{attribute 'linkalways'} 
{attribute 'no_explicit_call' := 'This FB is a CLASS and must be accessed using methods or properties'}
{attribute 'enable_dynamic_creation'}
FUNCTION_BLOCK FINAL NE_REAL EXTENDS Node
VAR
	in1 : _REAL(0.0);
	in2 : _REAL(0.0);
	out : _BOOL(FALSE);
END_VAR

METHOD PUBLIC Clone : I_Node
VAR
	pNode : POINTER TO NE_REAL;
END_VAR
pNode := __NEW(NE_REAL);
Clone := pNode^;
END_METHOD

METHOD FB_init : BOOL
VAR_INPUT
	bInitRetains : BOOL; // if TRUE, the retain variables are initialized (warm start / cold start)
	bInCopyCode : BOOL;  // if TRUE, the instance afterwards gets moved into the copy code (online change)
END_VAR
AddInput('in1',THIS^.in1);
AddInput('in2',THIS^.in2);
AddOutput('out', THIS^.out);
END_METHOD

METHOD PROTECTED OnExecute
VAR
END_VAR
out.Value := in1.Value <> in2.Value;
END_METHOD

END_FUNCTION_BLOCK

(* stored: Version 1.1.0.1, ProductVersion 3.1.4024.15
   POU NE_REAL: Id {a00dca68-9e9e-467b-a723-a2618a16da22}, SpecialFunc None
   Folder Constructor: Id {15e8fc73-f76e-45e3-9cc5-0c826013927e}
   Method Clone: Id {e5ce46a0-80d7-4106-a327-d2551ad97dd7}
   Method FB_init: Id {1b593138-0621-4288-906a-c8e7b4ae8038}
   Method OnExecute: Id {342a6d4d-c8a4-4f4f-8f1c-9d4dee35cd82} *)
